Fanuc KAREL source: kx00016.KL

-- PROVISIONAL review KL for V1013-1; original PC SHA256 583671f5aabab8a45f15359fd59945ef8815474244437ef1317031c998f5c5b2
-- Incomplete behavior may be omitted. Consult companion uncertainty JSON. Do not deploy.
PROGRAM KX00016
%NOLOCKGROUP
VAR
  I : INTEGER
  J : INTEGER
  B : BOOLEAN
  F : FILE
  S : STRING[80]
-- UNRESOLVED_DECL P type=000102
BEGIN
  -- UNRESOLVED_PC offsets 5-7; opcodes 9D,0D
  -- UNRESOLVED_PC offsets 12-16; opcodes 7F
END KX00016
